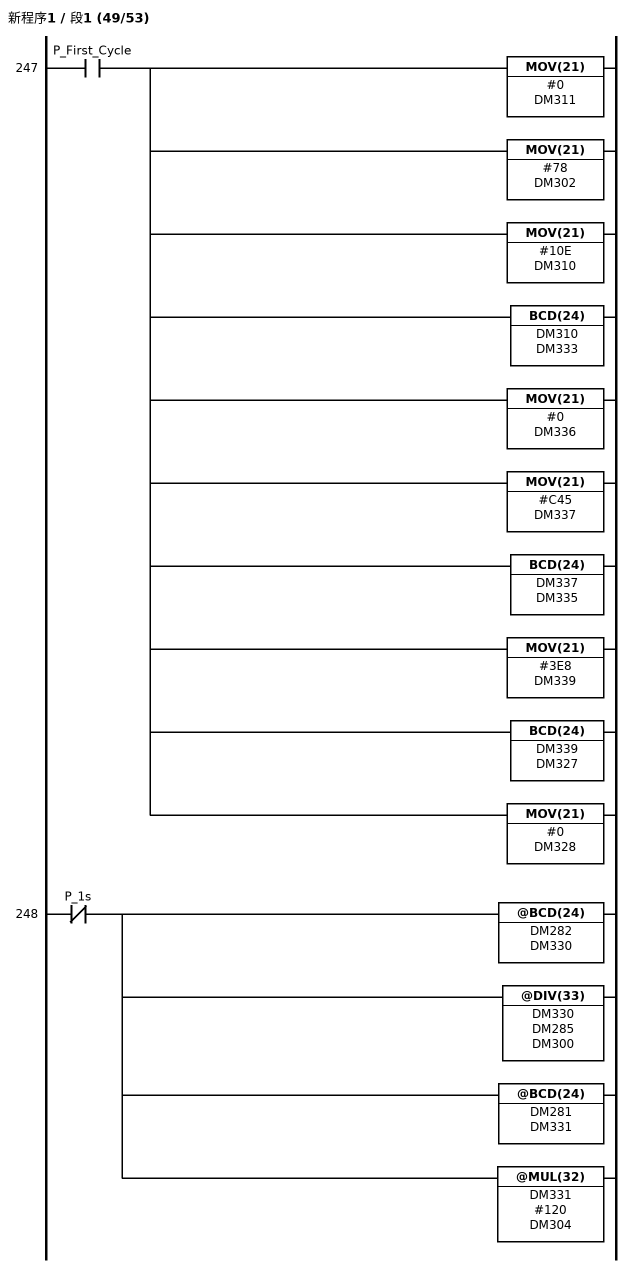
; [picture p48: 新程序1 / 段1, rungs 247-248]
; rung 247
LD P_First_Cycle
MOV(21) #0 DM311
MOV(21) #78 DM302
MOV(21) #10E DM310
BCD(24) DM310 DM333
MOV(21) #0 DM336
MOV(21) #C45 DM337
BCD(24) DM337 DM335
MOV(21) #3E8 DM339
BCD(24) DM339 DM327
MOV(21) #0 DM328
; rung 248
LDNOT P_1s
@BCD(24) DM282 DM330
@DIV(33) DM330 DM285 DM300
@BCD(24) DM281 DM331
@MUL(32) DM331 #120 DM304

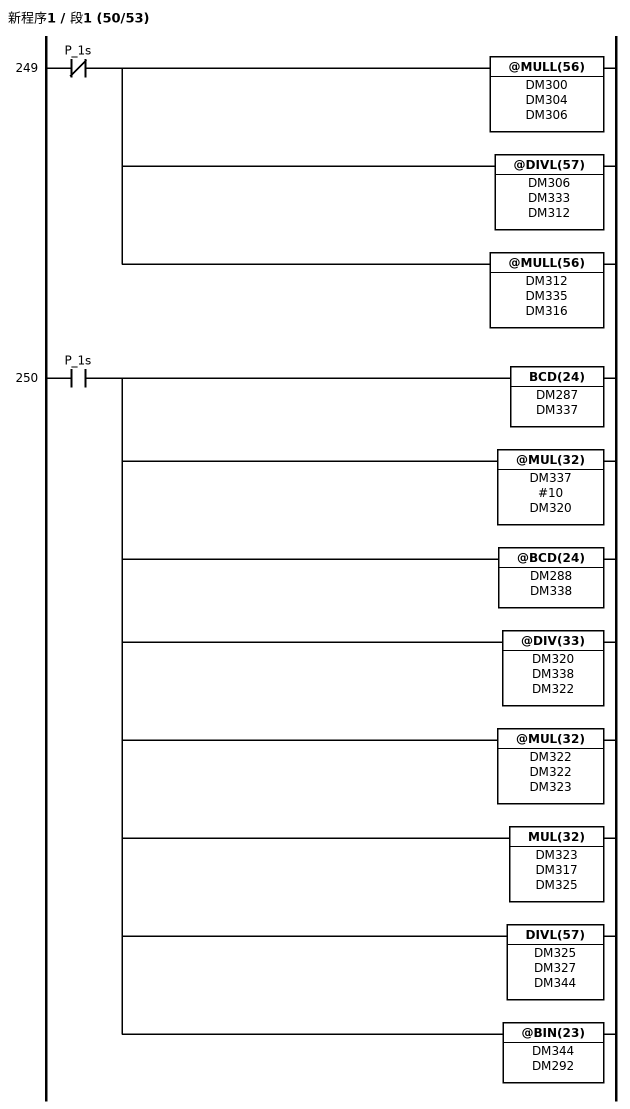
; rung 249
LDNOT P_1s
@MULL(56) DM300 DM304 DM306
@DIVL(57) DM306 DM333 DM312
@MULL(56) DM312 DM335 DM316
; rung 250
LD P_1s
BCD(24) DM287 DM337
@MUL(32) DM337 #10 DM320
@BCD(24) DM288 DM338
@DIV(33) DM320 DM338 DM322
@MUL(32) DM322 DM322 DM323
MUL(32) DM323 DM317 DM325
DIVL(57) DM325 DM327 DM344
@BIN(23) DM344 DM292

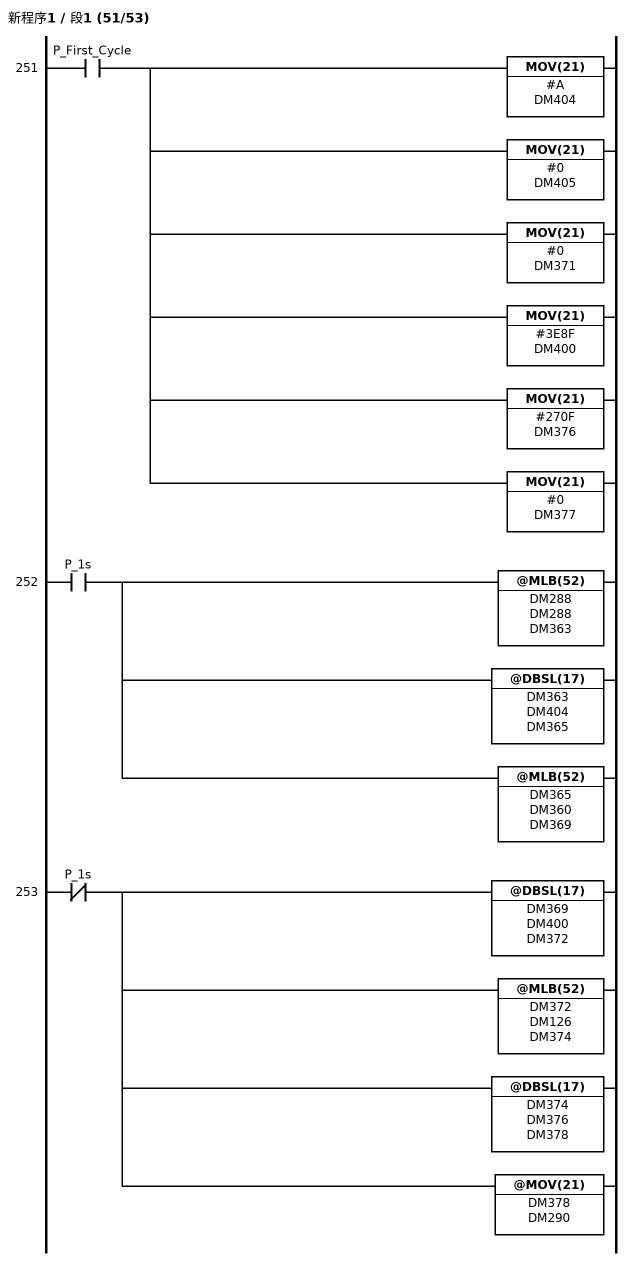
; rung 251
LD P_First_Cycle
MOV(21) #A DM404
MOV(21) #0 DM405
MOV(21) #0 DM371
MOV(21) #3E8F DM400
MOV(21) #270F DM376
MOV(21) #0 DM377
; rung 252
LD P_1s
@MLB(52) DM288 DM288 DM363
@DBSL(17) DM363 DM404 DM365
@MLB(52) DM365 DM360 DM369
; rung 253
LDNOT P_1s
@DBSL(17) DM369 DM400 DM372
@MLB(52) DM372 DM126 DM374
@DBSL(17) DM374 DM376 DM378
@MOV(21) DM378 DM290

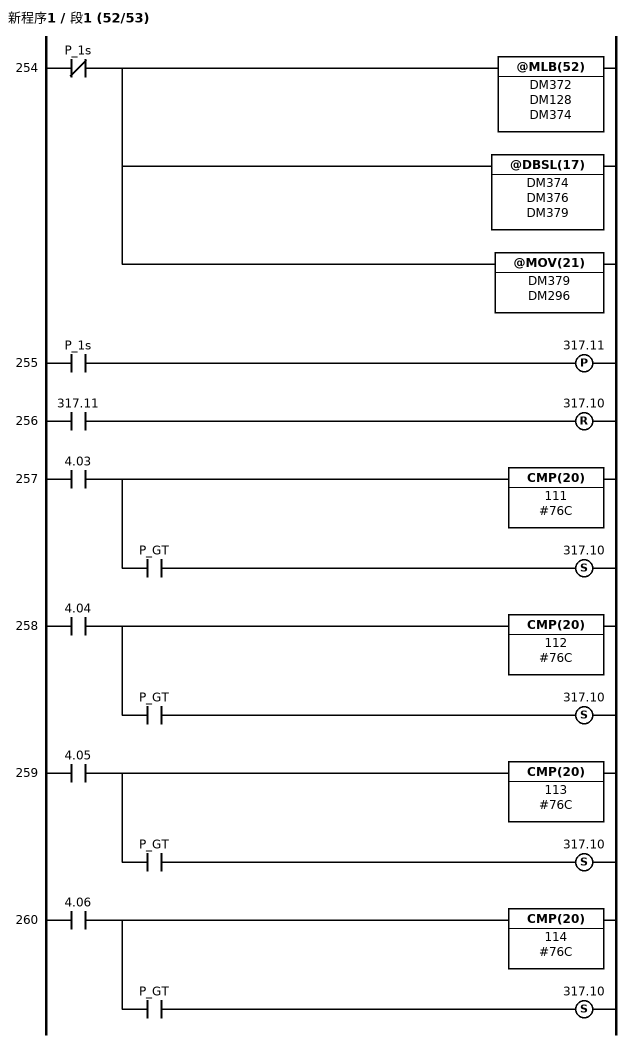
; rung 254
LDNOT P_1s
@MLB(52) DM372 DM128 DM374
@DBSL(17) DM374 DM376 DM379
@MOV(21) DM379 DM296
; rung 255
LD P_1s
DIFU(13) 317.11
; rung 256
LD 317.11
RSET 317.10
; rung 257
LD 4.03
CMP(20) 111 #76C
AND P_GT
SET 317.10
; rung 258
LD 4.04
CMP(20) 112 #76C
AND P_GT
SET 317.10
; rung 259
LD 4.05
CMP(20) 113 #76C
AND P_GT
SET 317.10
; rung 260
LD 4.06
CMP(20) 114 #76C
AND P_GT
SET 317.10

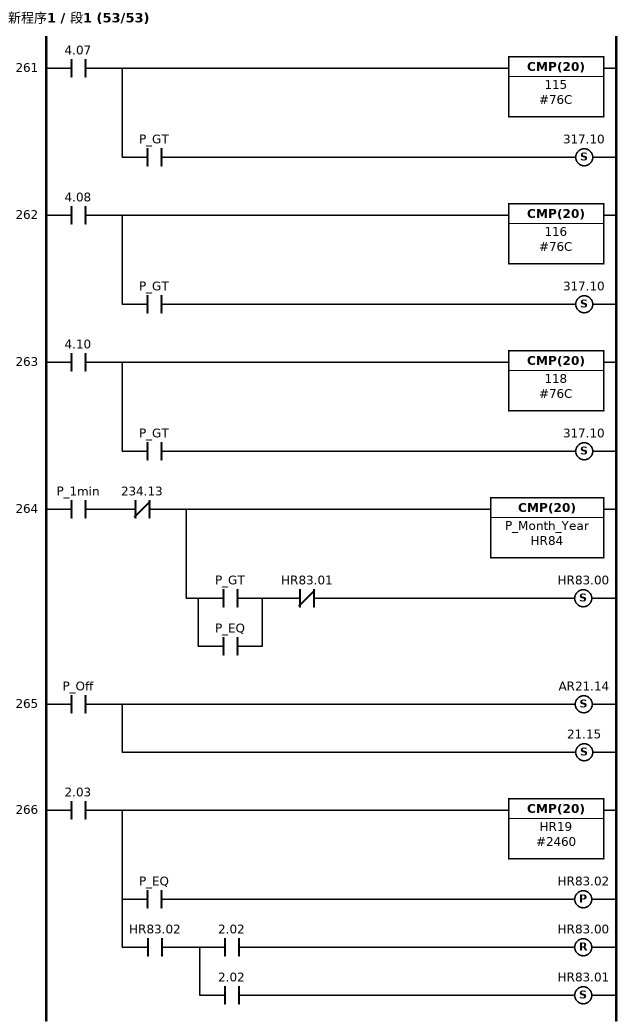
; rung 261
LD 4.07
CMP(20) 115 #76C
AND P_GT
SET 317.10
; rung 262
LD 4.08
CMP(20) 116 #76C
AND P_GT
SET 317.10
; rung 263
LD 4.10
CMP(20) 118 #76C
AND P_GT
SET 317.10
; rung 264
LD P_1min
ANDNOT 234.13
CMP(20) P_Month_Year HR84
LD P_GT
OR P_EQ
ANDNOT HR83.01
ANDLD
SET HR83.00
; rung 265
LD P_Off
SET AR21.14
SET 21.15
; rung 266
LD 2.03
OUT TR0
CMP(20) HR19 #2460
AND P_EQ
DIFU(13) HR83.02
LD TR0
AND HR83.02
OUT TR0
AND 2.02
RSET HR83.00
LD TR0
AND 2.02
SET HR83.01
; rung 267
END(01)